PROGRAM MAIN
VAR
	BOOL1 AT %MX0.0:BOOL;
	ib: INT;
	Tool1: TON;
	stat: BOOL;
	tt: BOOL;
	ss: BOOL;
	CTU1:CTU;
END_VAR

ib:=1;
Tool1(IN:= ss, PT:=t#3s , Q=> , ET=> );
CTU1(
	CU:= , 
	RESET:= , 
	PV:= , 
	Q=> , 
	CV=> );

END_PROGRAM

(* stored: Version 1.1.0.1, ProductVersion 3.1.4024.10
   POU MAIN: Id {9b790b26-15d0-458b-8eed-61ba45227661}, SpecialFunc None *)
